{attribute 'linkalways'} 
{attribute 'no_explicit_call' := 'This FB is a CLASS and must be accessed using methods or properties'}
{attribute 'enable_dynamic_creation'}
FUNCTION_BLOCK FINAL OR_ULINT EXTENDS Node
VAR
	in1 : _ULINT(0);
	in2 : _ULINT(0);
	out : _ULINT(0);
END_VAR

METHOD PUBLIC Clone : I_Node
VAR
	pNode : POINTER TO OR_ULINT;
END_VAR
pNode := __NEW(OR_ULINT);
Clone := pNode^;
END_METHOD

METHOD FB_init : BOOL
VAR_INPUT
	bInitRetains : BOOL; // if TRUE, the retain variables are initialized (warm start / cold start)
	bInCopyCode : BOOL;  // if TRUE, the instance afterwards gets moved into the copy code (online change)
END_VAR
AddInput('in1',THIS^.in1);
AddInput('in2',THIS^.in2);
AddOutput('out', THIS^.out);
END_METHOD

METHOD PROTECTED OnExecute
VAR
END_VAR
out.Value := in1.Value OR in2.Value;
END_METHOD

END_FUNCTION_BLOCK

(* stored: Version 1.1.0.1, ProductVersion 3.1.4024.15
   POU OR_ULINT: Id {16aeeb29-d5ee-48a0-a26e-77a2648b5248}, SpecialFunc None
   Folder Constructor: Id {a2eadc10-969a-439c-b452-86c2a44280ee}
   Method Clone: Id {ef6ec4be-9952-4fe1-a7ce-9c16cbc8af1d}
   Method FB_init: Id {6631a624-6511-469a-ba38-9f46bc07856d}
   Method OnExecute: Id {465b4e50-51d2-446c-9ea0-49a15645df5d} *)
